// TIA Portal V19 export
TYPE "UDT_EXPSM"
   STRUCT
      simvalue : Real := 0.0;   // Simulation value
      actual : Real := 0.0;   // Actual value
      output : Real := 0.0;   // Output value after smoothing (or not if disabled)
      "dt" : Real := 0.0;   // Dt in ms
      T { S7_SetPoint := 'True'} : Real := 0.0;   // Time to reach 63.2% = 1-1/e of original signal (must >=Dt)
      "a" : Real := 0.0;   // a = 1- e^(-Dt/T) and if Dt<<<T then a=Dt/T
      limit { S7_SetPoint := 'True'} : Real := 0.0;   // Limit near value that forces the Sn to break the loop and catch the Xn
      error : Bool := false;   // Out of limits
      simcmd : Bool := false;   // Simulation command
      exp_sm { S7_SetPoint := 'True'} : Bool := false;   // Exponential smoothing function (1=en, 0=dis)
      unit { S7_SetPoint := 'True'} : WString := WSTRING#'';   // Unit
   END_STRUCT;
END_TYPE
